SUBAPPLICATION Zaehler_Einsatzdauer (* Generischer persistenter Zaehler fuer die Einsatzdauer in Sekunden; rechnet den Zaehlerstand in Stunden/Minuten um, speichert beide Werte persistent im NVS und zeigt sie auf dem Terminal an *)
  (* Standard: 61499-2 *)
  (* Version 1.0, 2023-02-17, Franz *)
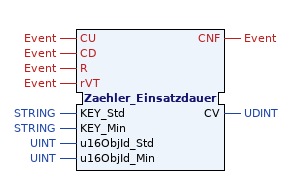
  EVENT_INPUT
    CU; (* Count Up *)
    CD; (* Count Down *)
    R; (* Reset *)
    rVT; (* refresh VT *)
  END_EVENT
  EVENT_OUTPUT
    CNF; (* Confirmation -- Counter Value was changed *)
  END_EVENT
  VAR_INPUT
    KEY_Std : STRING; (* NVS-Schluessel fuer den Stunden-Anteil der Einsatzdauer *)
    KEY_Min : STRING; (* NVS-Schluessel fuer den Minuten-Anteil der Einsatzdauer *)
    u16ObjId_Std : UINT; (* Objekt-ID des Zahlenwert-Objekts fuer die Stunden auf dem Terminal *)
    u16ObjId_Min : UINT; (* Objekt-ID des Zahlenwert-Objekts fuer die Minuten auf dem Terminal *)
  END_VAR
  VAR_OUTPUT
    CV : UDINT; (* Zaehlerstand in Sekunden (Rohwert des Zaehlers) *)
  END_VAR
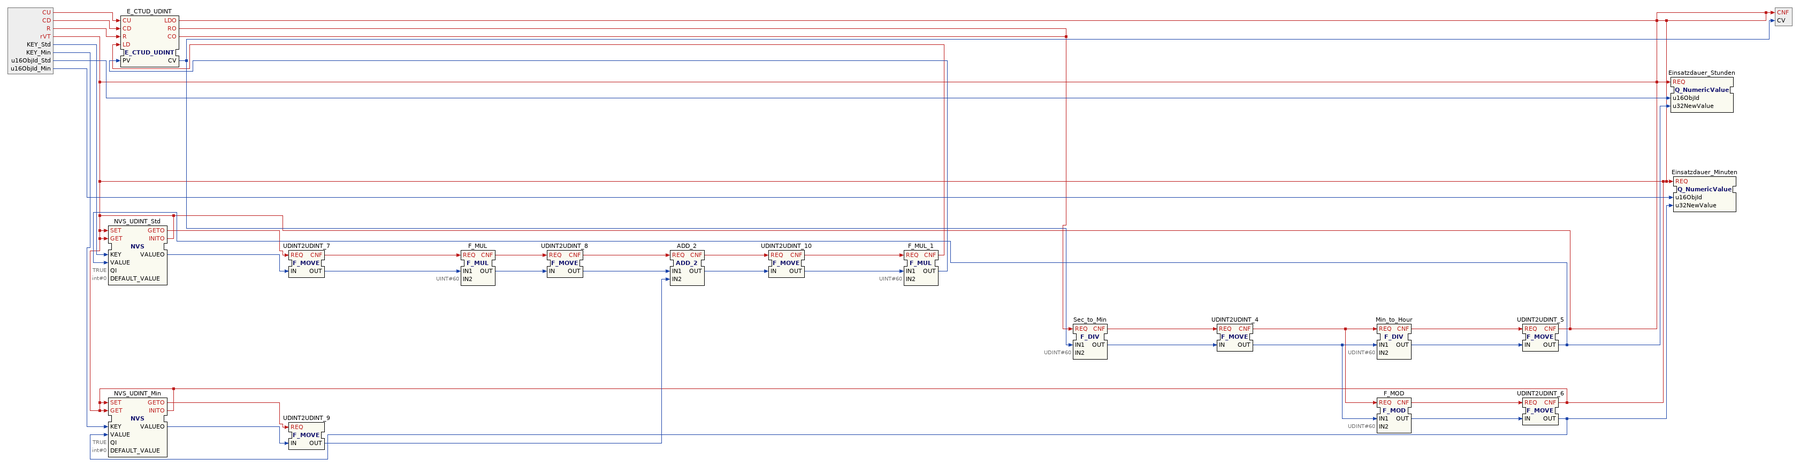
  FBS
    E_CTUD_UDINT : iec61499::events::E_CTUD_UDINT;
    Einsatzdauer_Stunden : isobus::UT::Q::Q_NumericValue;
    NVS_UDINT_Std : logiBUS::storage::esp32_nvs::NVS(QI := TRUE, DEFAULT_VALUE := int#0);
    UDINT2UDINT_4 : iec61131::selection::F_MOVE; {SET_ATTRIBUTE(DataType, UDINT)}
    F_MOD : iec61131::arithmetic::F_MOD(IN2 := UDINT#60);
    Min_to_Hour : iec61131::arithmetic::F_DIV(IN2 := UDINT#60);
    Sec_to_Min : iec61131::arithmetic::F_DIV(IN2 := UDINT#60);
    NVS_UDINT_Min : logiBUS::storage::esp32_nvs::NVS(QI := TRUE, DEFAULT_VALUE := int#0);
    Einsatzdauer_Minuten : isobus::UT::Q::Q_NumericValue;
    UDINT2UDINT_5 : iec61131::selection::F_MOVE; {SET_ATTRIBUTE(DataType, UDINT)}
    UDINT2UDINT_6 : iec61131::selection::F_MOVE; {SET_ATTRIBUTE(DataType, UDINT)}
    F_MUL : iec61131::arithmetic::F_MUL(IN2 := UINT#60);
    UDINT2UDINT_7 : iec61131::selection::F_MOVE; {SET_ATTRIBUTE(DataType, UDINT)}
    UDINT2UDINT_8 : iec61131::selection::F_MOVE; {SET_ATTRIBUTE(DataType, UDINT)}
    ADD_2 : iec61131::arithmetic::ADD_2;
    UDINT2UDINT_9 : iec61131::selection::F_MOVE; {SET_ATTRIBUTE(DataType, UDINT)}
    F_MUL_1 : iec61131::arithmetic::F_MUL(IN2 := UINT#60);
    UDINT2UDINT_10 : iec61131::selection::F_MOVE; {SET_ATTRIBUTE(DataType, UDINT)}
  END_FBS
  EVENT_CONNECTIONS
    CU TO E_CTUD_UDINT.CU;
    CD TO E_CTUD_UDINT.CD;
    R TO E_CTUD_UDINT.R;
    E_CTUD_UDINT.LDO TO CNF;
    UDINT2UDINT_4.CNF TO F_MOD.REQ;
    UDINT2UDINT_4.CNF TO Min_to_Hour.REQ;
    Min_to_Hour.CNF TO UDINT2UDINT_5.REQ;
    F_MOD.CNF TO UDINT2UDINT_6.REQ;
    UDINT2UDINT_5.CNF TO NVS_UDINT_Std.SET;
    UDINT2UDINT_6.CNF TO NVS_UDINT_Min.SET;
    E_CTUD_UDINT.LDO TO Einsatzdauer_Stunden.REQ;
    E_CTUD_UDINT.LDO TO Einsatzdauer_Minuten.REQ;
    UDINT2UDINT_5.CNF TO CNF;
    UDINT2UDINT_6.CNF TO Einsatzdauer_Minuten.REQ;
    UDINT2UDINT_5.CNF TO Einsatzdauer_Stunden.REQ;
    NVS_UDINT_Std.GETO TO UDINT2UDINT_7.REQ;
    UDINT2UDINT_7.CNF TO F_MUL.REQ;
    F_MUL.CNF TO UDINT2UDINT_8.REQ;
    UDINT2UDINT_8.CNF TO ADD_2.REQ;
    NVS_UDINT_Min.GETO TO UDINT2UDINT_9.REQ;
    E_CTUD_UDINT.RO TO Sec_to_Min.REQ;
    E_CTUD_UDINT.CO TO Sec_to_Min.REQ;
    ADD_2.CNF TO UDINT2UDINT_10.REQ;
    UDINT2UDINT_10.CNF TO F_MUL_1.REQ;
    F_MUL_1.CNF TO E_CTUD_UDINT.LD;
    Sec_to_Min.CNF TO UDINT2UDINT_4.REQ;
    rVT TO Einsatzdauer_Stunden.REQ;
    rVT TO Einsatzdauer_Minuten.REQ;
    NVS_UDINT_Std.INITO TO NVS_UDINT_Std.GET;
    NVS_UDINT_Min.INITO TO NVS_UDINT_Min.GET;
    rVT TO NVS_UDINT_Std.GET;
    rVT TO NVS_UDINT_Min.GET;
  END_CONNECTIONS
  DATA_CONNECTIONS
    E_CTUD_UDINT.CV TO CV;
    u16ObjId_Std TO Einsatzdauer_Stunden.u16ObjId;
    KEY_Std TO NVS_UDINT_Std.KEY;
    UDINT2UDINT_4.OUT TO Min_to_Hour.IN1;
    UDINT2UDINT_4.OUT TO F_MOD.IN1;
    KEY_Min TO NVS_UDINT_Min.KEY;
    u16ObjId_Min TO Einsatzdauer_Minuten.u16ObjId;
    Min_to_Hour.OUT TO UDINT2UDINT_5.IN;
    UDINT2UDINT_5.OUT TO NVS_UDINT_Std.VALUE;
    F_MOD.OUT TO UDINT2UDINT_6.IN;
    UDINT2UDINT_6.OUT TO NVS_UDINT_Min.VALUE;
    UDINT2UDINT_6.OUT TO Einsatzdauer_Minuten.u32NewValue;
    UDINT2UDINT_5.OUT TO Einsatzdauer_Stunden.u32NewValue;
    NVS_UDINT_Std.VALUEO TO UDINT2UDINT_7.IN;
    UDINT2UDINT_7.OUT TO F_MUL.IN1;
    F_MUL.OUT TO UDINT2UDINT_8.IN;
    UDINT2UDINT_8.OUT TO ADD_2.IN1;
    NVS_UDINT_Min.VALUEO TO UDINT2UDINT_9.IN;
    UDINT2UDINT_9.OUT TO ADD_2.IN2;
    E_CTUD_UDINT.CV TO Sec_to_Min.IN1;
    ADD_2.OUT TO UDINT2UDINT_10.IN;
    UDINT2UDINT_10.OUT TO F_MUL_1.IN1;
    F_MUL_1.OUT TO E_CTUD_UDINT.PV;
    Sec_to_Min.OUT TO UDINT2UDINT_4.IN;
  END_CONNECTIONS
END_SUBAPPLICATION
